TEXTLIST TextList_UpDownSlot_state
  0 = 'off'
  1 = 'up'
  2 = 'down'
  4 = 'waiting_up'
  5 = 'waiting_down'
  100 = 'error'
   = ''
END_TEXTLIST

(* stored: Version 1.1.0.1, ProductVersion 3.1.4024.11
   TextList TextList_UpDownSlot_state: Id {980e0561-f323-49d7-b7c1-3c425fe876a1} *)
